Universal Robots PolyScope program: happy_bday.urp

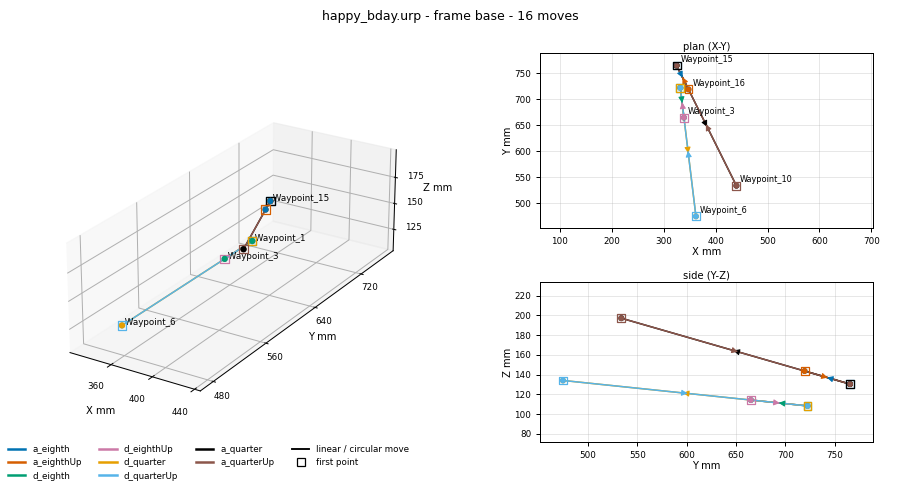
[picture p0: tool path of happy_bday.urp in frame base, 16 of 16 moves have a stored position in this frame; points joined in program order, loops and branches not executed]
Program happy_bday (installation=string_planes directory=/programs createdIn=5.17.3 lastSavedIn=5.17.3 robotSerialNumber=20245501435)
Calibrated DH parameters: a=[0.000154, -0.137004, -0.385524, -0.00002, 0.000092, 0]; d=[0.162441, 211.794786, -230.585024, 18.923638, 0.099786, 0.09951]; alpha=[1.569493, -0.001902, 0.003874, 1.570111, -1.570167, 0]; deltaTheta=[0, -1.242934, 1.056292, 0.186646, 0.000002, 0.000001]
InitVariablesNode
Robot Program (runOnlyOnce=false)
  Wait Sleep waitTime=10
  Call d_eighth
  Call d_eighthUp
  Call d_quarter
  Call d_quarterUp
  Call d_quarter
  Call d_quarterUp
  Wait Sleep waitTime=1
  Call d_eighth
  Call d_eighthUp
  Call d_quarter
  Call d_quarterUp
  Call a_quarter
  Call d_quarterUp
  Wait Sleep waitTime=1
  Call d_eighth
  Call d_eighthUp
  Call a_quarter
  Call a_quarterUp
  Call d_quarter
  Call d_quarterUp
  Call d_quarter
  Call a_quarterUp
  Call a_quarter
  Call d_quarterUp
  Call a_quarter
  Call d_quarterUp
  Wait Sleep waitTime=2
SubProgram a_eighth (keepSynchronizedWithDisk=false) programFile=/programs/a_eighth.urp
  MoveL speed 250 mm/s, acceleration 1200 mm/s^2 (useActiveTCP=true) feature=Plane_1
    Waypoint Waypoint_15: TCP in base x=324.752 y=765.324 z=130.385 mm, rx=-1.4944 ry=-2.2778 rz=1.1569 rad; joints [-127.056, -14.742, 33.541, -62.028, -82.973, -153.445] deg; TCP offset x=28.21 y=-96.107 z=-99.69 mm, rx=0 ry=0 rz=0 rad; feature pose in base x=325.716 y=793.387 z=118.207 mm, rx=-2.2082 ry=-0.2474 rz=-1.9195 rad
    Waypoint Waypoint_16: TCP in base x=347.657 y=719.315 z=143.639 mm, rx=-1.4944 ry=-2.2778 rz=1.1569 rad; joints [-130.247, -21.46, 45.573, -67.125, -85.28, -155.63] deg; feature pose in base x=325.716 y=793.387 z=118.207 mm, rx=-2.2082 ry=-0.2474 rz=-1.9195 rad
SubProgram a_eighthUp (keepSynchronizedWithDisk=false) programFile=/programs/a_eighthUp.urp
  MoveL speed 250 mm/s, acceleration 1200 mm/s^2 (useActiveTCP=true) feature=Plane_1
    Waypoint Waypoint_13: TCP in base x=347.657 y=719.315 z=143.639 mm, rx=-1.4944 ry=-2.2778 rz=1.1569 rad; joints [-130.247, -21.46, 45.573, -67.125, -85.28, -155.63] deg
    Waypoint Waypoint_14: TCP in base x=324.752 y=765.324 z=130.385 mm, rx=-1.4944 ry=-2.2778 rz=1.1569 rad; joints [-127.056, -14.742, 33.541, -62.028, -82.973, -153.445] deg; feature pose in base x=325.716 y=793.387 z=118.207 mm, rx=-2.2082 ry=-0.2474 rz=-1.9195 rad
SubProgram -> a_quarterUp
SubProgram -> a_quarter
SubProgram -> d_quarterUp
SubProgram -> d_quarter
SubProgram -> d_eighthUp
SubProgram -> d_eighth
SubProgram d_eighth (keepSynchronizedWithDisk=false) programFile=/programs/d_eighth.urp
  MoveL speed 250 mm/s, acceleration 1200 mm/s^2 (useActiveTCP=true) feature=Plane_2
    Waypoint Waypoint_1: TCP in base x=331.971 y=722.315 z=108.291 mm, rx=-1.645 ry=-2.1081 rz=1.0591 rad; joints [-129.709, -21.469, 51.981, -76.268, -76.862, -148.975] deg; feature pose in base x=343.605 y=747.803 z=100.778 mm, rx=2.7685 ry=0.1285 rz=1.3673 rad
    Waypoint Waypoint_3: TCP in base x=338.919 y=665.001 z=114.26 mm, rx=-1.6378 ry=-2.1148 rz=1.0804 rad; joints [-132.848, -27.946, 64.83, -81.449, -79.739, -151.46] deg; feature pose in base x=343.605 y=747.803 z=100.778 mm, rx=2.7685 ry=0.1285 rz=1.3673 rad
SubProgram d_eighthUp (keepSynchronizedWithDisk=false) programFile=/programs/d_eighthUp.urp
  MoveL speed 250 mm/s, acceleration 1200 mm/s^2 (useActiveTCP=true) feature=Plane_2
    Waypoint Waypoint_2: TCP in base x=338.919 y=665.001 z=114.26 mm, rx=-1.6378 ry=-2.1148 rz=1.0804 rad; joints [-132.848, -27.946, 64.83, -81.449, -79.739, -151.46] deg; feature pose in base x=343.605 y=747.803 z=100.778 mm, rx=2.7685 ry=0.1285 rz=1.3673 rad
    Waypoint Waypoint_4: TCP in base x=331.971 y=722.315 z=108.291 mm, rx=-1.645 ry=-2.1081 rz=1.0591 rad; joints [-129.709, -21.469, 51.981, -76.268, -76.862, -148.975] deg
SubProgram d_quarter (keepSynchronizedWithDisk=false) programFile=/programs/d_quarter.urp
  MoveL speed 250 mm/s, acceleration 1200 mm/s^2 (useActiveTCP=true) feature=Plane_2
    Waypoint Waypoint_5: TCP in base x=331.971 y=722.315 z=108.291 mm, rx=-1.645 ry=-2.1081 rz=1.0591 rad; joints [-129.709, -21.469, 51.981, -76.268, -76.862, -148.975] deg
    Waypoint Waypoint_6: TCP in base x=362.01 y=474.766 z=134.068 mm, rx=-1.613 ry=-2.1363 rz=1.1513 rad; joints [-146.069, -43.376, 94.489, -92.87, -91.874, -160.9] deg; feature pose in base x=343.605 y=747.803 z=100.778 mm, rx=2.7685 ry=0.1285 rz=1.3673 rad
SubProgram d_quarterUp (keepSynchronizedWithDisk=false) programFile=/programs/d_quarterUp.urp
  MoveL speed 250 mm/s, acceleration 1200 mm/s^2 (useActiveTCP=true) feature=Plane_2
    Waypoint Waypoint_7: TCP in base x=362.01 y=474.766 z=134.068 mm, rx=-1.613 ry=-2.1363 rz=1.1513 rad; joints [-146.069, -43.376, 94.489, -92.87, -91.874, -160.9] deg; feature pose in base x=343.605 y=747.803 z=100.778 mm, rx=2.7685 ry=0.1285 rz=1.3673 rad
    Waypoint Waypoint_8: TCP in base x=331.971 y=722.315 z=108.291 mm, rx=-1.645 ry=-2.1081 rz=1.0591 rad; joints [-129.709, -21.469, 51.981, -76.268, -76.862, -148.975] deg; feature pose in base x=343.605 y=747.803 z=100.778 mm, rx=2.7685 ry=0.1285 rz=1.3673 rad
SubProgram a_quarter (keepSynchronizedWithDisk=false) programFile=/programs/a_quarter.urp
  MoveL speed 250 mm/s, acceleration 1200 mm/s^2 (useActiveTCP=true) feature=Plane_1
    Waypoint Waypoint_9: TCP in base x=324.752 y=765.324 z=130.385 mm, rx=-1.4944 ry=-2.2778 rz=1.1569 rad; joints [-127.056, -14.742, 33.541, -62.028, -82.973, -153.445] deg; feature pose in base x=325.716 y=793.387 z=118.207 mm, rx=-2.2082 ry=-0.2474 rz=-1.9195 rad
    Waypoint Waypoint_10: TCP in base x=439.971 y=533.839 z=197.07 mm, rx=-1.4944 ry=-2.2778 rz=1.1569 rad; joints [-144.985, -38.317, 71.569, -76.412, -96.031, -165.68] deg; feature pose in base x=325.716 y=793.387 z=118.207 mm, rx=-2.2082 ry=-0.2474 rz=-1.9195 rad
SubProgram a_quarterUp (keepSynchronizedWithDisk=false) programFile=/programs/a_quarterUp.urp
  MoveL speed 250 mm/s, acceleration 1200 mm/s^2 (useActiveTCP=true) feature=Plane_1
    Waypoint Waypoint_11: TCP in base x=439.971 y=533.839 z=197.07 mm, rx=-1.4944 ry=-2.2778 rz=1.1569 rad; joints [-144.985, -38.317, 71.569, -76.412, -96.031, -165.68] deg; feature pose in base x=325.716 y=793.387 z=118.207 mm, rx=-2.2082 ry=-0.2474 rz=-1.9195 rad
    Waypoint Waypoint_12: TCP in base x=324.752 y=765.324 z=130.385 mm, rx=-1.4944 ry=-2.2778 rz=1.1569 rad; joints [-127.056, -14.742, 33.541, -62.028, -82.973, -153.445] deg; feature pose in base x=325.716 y=793.387 z=118.207 mm, rx=-2.2082 ry=-0.2474 rz=-1.9195 rad
